TYPE AX5000_S_0109 :
STRUCT
	Motor_peak_current:UDINT;
END_STRUCT
END_TYPE

(* stored: Version 1.1.0.1, ProductVersion 3.1.4024.3
   DUT AX5000_S_0109: Id {7046b3e5-9947-448c-87a3-039697366161} *)
